(* PLC project Generated.project, CODESYS CODESYS V3.5 SP19 Patch 1 *)
(* stored: creationDateTime 2026-08-30T23:29:56.443516, modificationDateTime 2026-08-30T23:29:56.443516 *)

(* ======================================================================= ST_fbDiveSearch_Outputs - Bus de sortie du cycle FB_DiveSearch ======================================================================= *)
TYPE ST_fbDiveSearch_Outputs : STRUCT
  StepState : E_DiveSearchState;  (* === ETAT DU CYCLE === Etape courante *)
  StepAtFault : E_DiveSearchState;  (* Etape figee au defaut *)
  DescendPermit : BOOL;  (* === PERMIS & ORDRES ASSISTES === Autorisation de descente assistee *)
  KoboldContactorCmd : BOOL;  (* Commande alimentation Kobold (fail-safe, coupe au front de fond) *)
  BottomTouchConfirmed : BOOL;  (* Fond confirme *)
  MinStepDown : INT;  (* Plancher palier descente *)
  OperatorActionId : WORD;  (* === DIAGNOSTIC OPERATEUR === Identifiant numerique de l'action *)
  OperatorAction : STRING(120);  (* Consigne operateur ASCII *)
END_STRUCT;
END_TYPE

(* values of E_DiveSearchState: WAIT_PRECONDITIONS: Attente benne ouverte, positions et Kobold au repos; READY_TO_DESCEND: Prêt à assister une demande de descente; SEARCHING_IMMERSION: Descending : attente front 0->1 dans fenêtre eau; SEARCHING_BOTTOM: Immersion validée : attente front 1->0 au fond; BOTTOM_CONFIRMED: Fond validé ; extraction peut être demandée; ERROR_HOLD: Séquence invalide, descente assistée interdite *)

{attribute 'qualified_only'}
{attribute 'strict'}
TYPE E_DiveSearchState : (WAIT_PRECONDITIONS := 0, READY_TO_DESCEND := 1, SEARCHING_IMMERSION := 2, SEARCHING_BOTTOM := 3, BOTTOM_CONFIRMED := 4, ERROR_HOLD := 5);
END_TYPE
